FUNCTION_BLOCK FB_TcBSD_Sendmail
VAR_INPUT
END_VAR
VAR_OUTPUT
END_VAR
VAR
//SMTP Sendmail
	fbMailSend:NT_StartProcess;			//Send Mail
	
//Mail Sendstring
	sCommand:STRING(512);			//Send Command
	
//Execute Send
	bProcessExecute:BOOL;					//Send Execute
	bProcessActive:BOOL;					//Send Active
	bProcessBusy:BOOL;						//Send Busy
	bProcessError:BOOL;					//Send Error
	
//Mail Parameter
	sAddressTO:STRING;					//Mail TO
	sAddressFROM:STRING;				//Mail FROM
	sAddressCC:STRING;					//Mail CC
	sAddressBCC:STRING;					//Mail BCC
	sMailMessage:STRING(255);			//Mail Message
	sMailSubject:STRING;				//Mail Subject
	
//Status & Helper
	tonExecuteReset: TON;				//Timer Execute Reset
		
END_VAR

(*

-Send Mail with /usr/bin/mail
-Installed ssmtp package required
-v0.1

*)

PROPERTY AddressBCC : STRING
SET
sAddressBCC:=AddressBCC;
END_SET
END_PROPERTY

PROPERTY AddressCC : STRING
SET
sAddressCC:=AddressCC;
END_SET
END_PROPERTY

PROPERTY AddressFROM : STRING
SET
sAddressFROM := AddressFROM;
END_SET
END_PROPERTY

PROPERTY AddressTO : STRING
SET
sAddressTO := AddressTO;
END_SET
END_PROPERTY

METHOD PRIVATE BuildCommand : INT
VAR_INPUT
END_VAR
//Build Sendstring
sCommand:= '"echo -e ';
sCommand:=CONCAT(sCommand, '\"');
sCommand:=CONCAT(sCommand, sMailMessage);
sCommand:=CONCAT(sCommand, '\"');
sCommand:=CONCAT(sCommand, ' | ');
sCommand:=CONCAT(sCommand, 'mail -s ');
sCommand:=CONCAT(sCommand, '\"');
sCommand:=CONCAT(sCommand, sMailSubject);
sCommand:=CONCAT(sCommand, '\"');
sCommand:=CONCAT(sCommand, ' ');
sCommand:=CONCAT(sCommand, sAddressTO);
IF sAddressCC <> '' THEN
	sCommand:=CONCAT(sCommand, ' -c ');
	sCommand:=CONCAT(sCommand, sAddressCC);
END_IF
IF sAddressBCC <> '' THEN
	sCommand:=CONCAT(sCommand, ' -b ');
	sCommand:=CONCAT(sCommand, sAddressBCC);
END_IF
sCommand:=CONCAT(sCommand, ' -F');
sCommand:=CONCAT(sCommand, '\"');
sCommand:=CONCAT(sCommand, sAddressFROM);
sCommand:=CONCAT(sCommand, '\"');
sCommand:=CONCAT(sCommand, '"');
END_METHOD

METHOD Cyclic : INT
VAR_INPUT
END_VAR
(*

--Call Cyclic

*)

//Send Mail
fbMailSend(
	NETID:= '', 
	PATHSTR:='/bin/sh -c' , 
	DIRNAME:='/bin' , 
	COMNDLINE:=sCommand , 
	START:=bProcessActive, 
	TMOUT:= , 
	BUSY=> , 
	ERR=> , 
	ERRID=> );

//Send Execute Reset		
tonExecuteReset(IN:=bProcessExecute=FALSE AND bProcessActive=TRUE , PT:=T#5S);
IF tonExecuteReset.Q THEN
	bProcessActive:=FALSE;
END_IF
bProcessExecute:=FALSE;

//Status Signals
bProcessBusy:=bProcessActive;
IF bProcessActive AND fbMailSend.ERR THEN
	bProcessError:=TRUE;
END_IF
END_METHOD

METHOD PUBLIC Execute : INT
VAR_INPUT
END_VAR
//Send Mail

//Build Sendstring
BuildCommand();

//Flag Securtiy
if bProcessExecute=false then
	bProcessActive:=TRUE;
	bProcessError:=FALSE;
END_IF
bProcessExecute:=TRUE;
END_METHOD

PROPERTY MailMessage : STRING (255)
SET
sMailMessage:=MailMEssage;
END_SET
END_PROPERTY

PROPERTY MailSubject : STRING
SET
sMailSubject:=MailSubject;
END_SET
END_PROPERTY

PROPERTY SendCommand : STRING(255)
GET
SendCommand:=sCommand;
END_GET
END_PROPERTY

END_FUNCTION_BLOCK

(* stored: Version 1.1.0.1, ProductVersion 3.1.4024.12
   POU FB_TcBSD_Sendmail: Id {5981f3e6-1b40-4ab6-b64e-0c06599d6540}, SpecialFunc None
   Property AddressBCC: Id {fd6b1475-6a8d-4b95-9e00-b18ae9fe83cb}
   Set Set: Id {c9874781-8fc7-45bb-a89e-2b900cccfdbd}
   Property AddressCC: Id {26955842-6288-432a-a9bb-343ef410393a}
   Set Set: Id {a742275a-a64a-4feb-a970-4caad40b24c5}
   Property AddressFROM: Id {a1fc6a04-97af-4fb9-acb1-cceaa5def81a}
   Set Set: Id {921b768a-c29f-4c04-a43b-c56632cdc521}
   Property AddressTO: Id {dfece2c1-9200-4dd8-a86a-749a3ed46bdf}
   Set Set: Id {7d829ad5-f517-45bf-abd0-c16f49eee572}
   Method BuildCommand: Id {41084b91-bdc1-4f00-a69f-c784fcee5b00}
   Method Cyclic: Id {2847d448-3c51-4961-b3af-fa158c7b4b6b}
   Method Execute: Id {bc93429f-fb74-46ec-ac1f-44d9099960bb}
   Property MailMessage: Id {0f383fe0-337d-46ac-8ef7-894a4a60962d}
   Set Set: Id {72348338-a4bf-48a5-9eac-954ebcb752d0}
   Property MailSubject: Id {4332c76f-788f-4e8c-962e-900c98b5af72}
   Set Set: Id {60e9fb6e-23f5-41fd-9a91-9407ed05b982}
   Property SendCommand: Id {c6b87f4b-d6e9-4c36-a5d3-3303a34998d0}
   Get Get: Id {a19136b8-7443-4464-905e-6ff259b3f968} *)
